{attribute 'GeneratedUsingTerminal: ER6001-0002-0016'}
{attribute addProperty BoxType "ER6001-0002-0016"}
{attribute addProperty Id "EtcSlaveTerminalBaseCOM_InputsAT %I*COM_Inputs_6C2FC20224COM_OutputsAT %Q*COM_Outputs_5D00B5E724WcStateAT %I*WcState_9091E0EB2InfoDataAT %I*InfoData_32EB74EA10"}
{attribute addProperty CRC "3110463989"}
{attribute addProperty Size "60"}
TYPE ER6001_B965E9F5 EXTENDS EtcSlaveTerminalBase :
STRUCT
	{attribute addProperty Name "COM_Inputs"}
	COM_Inputs : COM_Inputs_6C2FC202;
	{attribute addProperty Name "COM_Outputs"}
	COM_Outputs : COM_Outputs_5D00B5E7;
	{attribute addProperty Name "WcState"}
	WcState : WcState_9091E0EB;
	{attribute addProperty Name "InfoData"}
	InfoData : InfoData_32EB74EA;
END_STRUCT
END_TYPE

(* stored: Version 1.2.0.0, ProductVersion 3.1.4024.9
   DUT ER6001_B965E9F5: Id {258e3d0a-46ba-4ea0-b033-18e679f2ef6b} *)
